// TIA Portal V18 export
VAR_GLOBAL   // PLC tag table "Table de variables_MODBUS_Client"
   MB_CLIENT_MODE AT %MB301 : USInt;   // Comment 1
   MB_DATA_ADDR AT %MD302 : UDInt;   // Comment 2
   MB_DATA_LEN AT %MW306 : UInt;   // Comment 3
   MB_CLIENT_REQ AT %M300.0 : Bool;   // Comment 4
   MB_CLIENT_DISC AT %M300.1 : Bool;   // Comment 5
   "Clock_0.5Hz" AT %M0.7 : Bool;
   AlwaysFALSE AT %M1.3 : Bool;
   AlwaysTRUE AT %M1.2 : Bool;
   "Clock_0.625Hz" AT %M0.6 : Bool;
   "Clock_1.25Hz" AT %M0.4 : Bool;
   Clock_1Hz AT %M0.5 : Bool;
   "Clock_2.5Hz" AT %M0.2 : Bool;
   Clock_2Hz AT %M0.3 : Bool;
   Clock_5Hz AT %M0.1 : Bool;
   Clock_10Hz AT %M0.0 : Bool;
   Clock_Byte AT %MB0 : Byte;
   DiagStatusUpdate AT %M1.1 : Bool;
   FirstScan AT %M1.0 : Bool;
   Cause_1 AT %M200.0 : Bool;
   Effect1 AT %M200.1 : Bool;
END_VAR
